// TIA Portal project "Parkplatz_1" (V20)

(* hardware
DEVICE "S7-1500/ET200MP-Station_1"  S7-1500 station
   slot 0: "Profilschiene_0"  Rack  6ES7 590-1***0-0AA0
   slot 1: "PLC_1"  CPU 1513-1 PN  6ES7 513-1AM03-0AB0  V4.0
      slot 3: "CPU-Display_1"  6ES7591-1AA00-0AA0
      slot 32768: "PROFINET-Schnittstelle_1"  X1
         slot 32769: "Port_1"  X1 P1
         slot 32770: "Port_2"  X1 P2
      slot 34817: "Virtual CP interface port_1"  Virtual CP interface port  Virtual CP interface port FW V4.0
   slot 2: "DI 16x24VDC BA_1"  DI 16x24VDC BA  6ES7 521-1BH10-0AA0  V1.1
   slot 3: "DQ 16x24VDC/0.5A ST_1"  DQ 16x24VDC/0.5A ST  6ES7 522-1BH00-0AB0  V2.0
   slot 4: "AI 8xU/I/R/RTD BA_1"  AI 8xU/I/R/RTD BA  6ES7 531-7QF00-0AB0  V1.0
   slot 5: "AQ 8xU/I HS_1"  AQ 8xU/I HS  6ES7 532-5HF00-0AB0  V2.2
   slot 6: "AQ 2xU/I ST_1"  AQ 2xU/I ST  6ES7 532-5NB00-0AB0  V1.0
*)

// ===== PLC "PLC_1"  CPU 1513-1 PN =====

VAR_GLOBAL   // PLC tag table "Standard-Variablentabelle"
   "PlcLabConnectIn01" AT %ID32760 : DWord;
   "PlcLabConnectIn02" AT %ID32764 : DWord;
   "PlcLabConnectOut01" AT %QD32760 : DWord;
   "PlcLabConnectOut02" AT %QD32764 : DWord;
   "Auto_rein_1" AT %M1.0 : Bool;
   "Auto_raus_1" AT %M1.1 : Bool;
   "Kein_Platz_frei" AT %M1.4 : Bool;
   "E1_Schranke_zu" AT %M2.0 : Bool;
   "A1_Schranke_zu" AT %M2.1 : Bool;
   "Plaetze_frei" AT %M1.5 : Bool;
   "Auto_raus_2" AT %M1.3 : Bool;
   "Auto_rein_2" AT %M1.2 : Bool;
   "E2_Schranke_zu" AT %M2.2 : Bool;
   "A2_Schranke_zu" AT %M2.3 : Bool;
END_VAR

VAR_GLOBAL   // PLC tag table "Eingänge"
   "B1" AT %E0.0 : Bool;   // Sensor 1 Einfahrt
   "B2" AT %E0.1 : Bool;   // Sensor 1 Ausfahrt
   "B3" AT %E0.2 : Bool;   // Sensor 2 Einfahrt
   "B4" AT %E0.3 : Bool;   // Sensor 2 Ausfahrt
   "S1" AT %E0.4 : Bool;   // Betriebsschalter
END_VAR

VAR_GLOBAL   // PLC tag table "Ausgänge"
   "P1" AT %A0.0 : Bool;   // Ampel 1 (rot)
   "P2" AT %A0.1 : Bool;   // Ampel 1 (grün)
   "P5" AT %AW32 : Int;   // Anzeige "Freie Parkplätze"
   "P6" AT %A0.4 : Bool;   // Schranke 1 Einfahrt
   "P7" AT %A0.5 : Bool;   // Schranke 1 Ausfahrt
   "P3" AT %A0.2 : Bool;   // Ampel 2 (rot)
   "P4" AT %A0.3 : Bool;   // Ampel 2 (grün)
   "P8" AT %A0.6 : Bool;   // Schranke 2 Einfahrt
   "P9" AT %A0.7 : Bool;   // Schranke 2 Ausfahrt
END_VAR

// folder: System blocks/Program resources

DATA_BLOCK "IEC_Counter_0_DB"   // DB1
{ S7_Optimized_Access := 'TRUE' }
AUTHOR : Simatic
FAMILY : IEC
NAME : CNTR
VERSION : 1.0
// stored: InstanceOfName IEC_COUNTER
"IEC_COUNTER"
BEGIN
   PV := 16;
END_DATA_BLOCK

DATA_BLOCK "IEC_Timer_0_DB"   // DB2
{ S7_Optimized_Access := 'TRUE' }
AUTHOR : Simatic
FAMILY : IEC
NAME : IEC_TMR
VERSION : 1.0
// stored: InstanceOfName IEC_TIMER
"IEC_TIMER"
BEGIN
END_DATA_BLOCK

DATA_BLOCK "IEC_Timer_0_DB_1"   // DB3
{ S7_Optimized_Access := 'TRUE' }
AUTHOR : Simatic
FAMILY : IEC
NAME : IEC_TMR
VERSION : 1.0
// stored: InstanceOfName IEC_TIMER
"IEC_TIMER"
BEGIN
END_DATA_BLOCK

DATA_BLOCK "IEC_Timer_0_DB_2"   // DB4
{ S7_Optimized_Access := 'TRUE' }
AUTHOR : Simatic
FAMILY : IEC
NAME : IEC_TMR
VERSION : 1.0
// stored: InstanceOfName IEC_TIMER
"IEC_TIMER"
BEGIN
END_DATA_BLOCK

DATA_BLOCK "IEC_Timer_0_DB_3"   // DB5
{ S7_Optimized_Access := 'TRUE' }
AUTHOR : Simatic
FAMILY : IEC
NAME : IEC_TMR
VERSION : 1.0
// stored: InstanceOfName IEC_TIMER
"IEC_TIMER"
BEGIN
END_DATA_BLOCK

// folder: (top level)

FUNCTION "Parkplatzsteuerung" : Void   // FC1, FBD
{ S7_Optimized_Access := 'TRUE' }
VERSION : 0.1
   VAR_TEMP   // added for the SCL form of the ladder/FBD networks
      _w1 : Bool;
      _w2 : Bool;
      _w3 : Bool;
      _w4 : Bool;
   END_VAR
BEGIN

REGION Network 1: Freie Plätze Zähler
   // Mithilfe des CTUD wird die Anzahl der freien Parkplätze gezählt. Über den Sensor B1 wird gezählt wenn ein Fahrzeug den Parkplatz betritt, dadurch gibt es einen freien Platz weniger. Über B2 wird gezählt wenn ein Fahrzeug den Parkplatz verlässt, dadurch gibt es einen freien Platz mehr. Die Grenze PV liegt auf 1, damit der Merker "Kein Platz frei" darunter auf FALSE geht. Bei 1 oder mehr gibt es freie Plätze, somit wird der Merker "Plätze frei" TRUE.
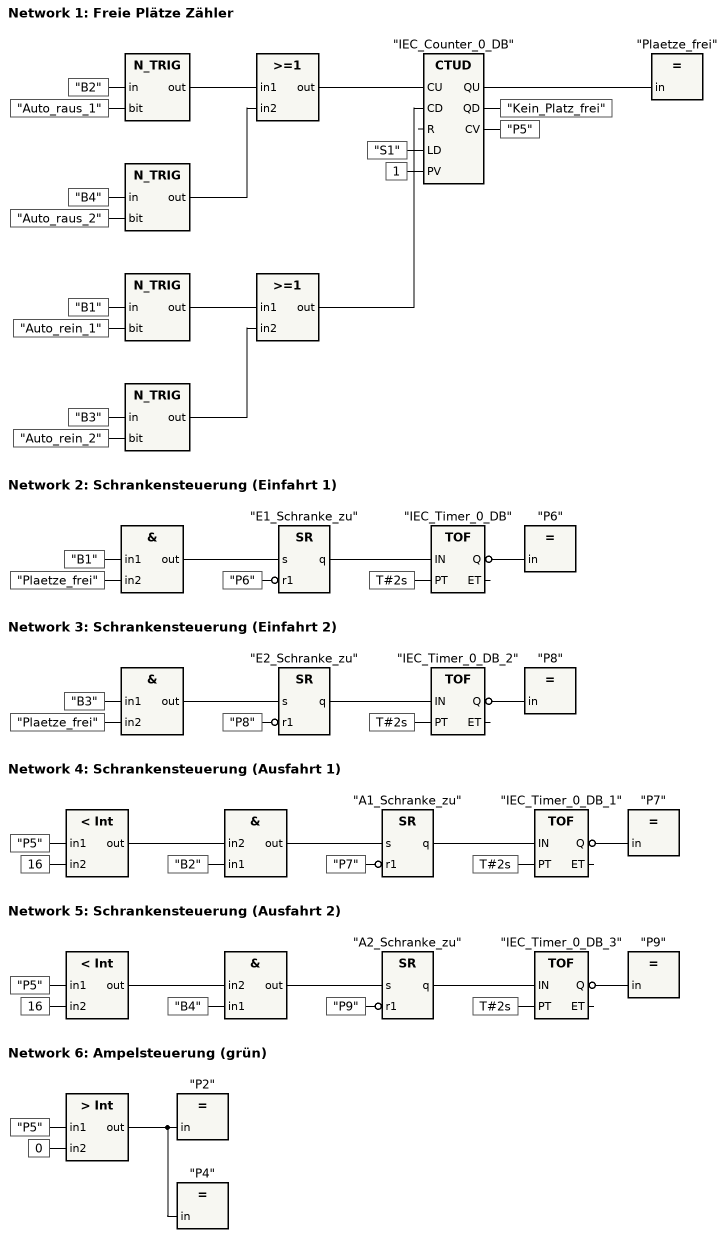
   #_w1 := NOT "B2" AND "Auto_raus_1";   // falling edge
   "Auto_raus_1" := "B2";
   #_w2 := NOT "B4" AND "Auto_raus_2";   // falling edge
   "Auto_raus_2" := "B4";
   #_w3 := NOT "B1" AND "Auto_rein_1";   // falling edge
   "Auto_rein_1" := "B1";
   #_w4 := NOT "B3" AND "Auto_rein_2";   // falling edge
   "Auto_rein_2" := "B3";
   "IEC_Counter_0_DB".CTUD(CU := #_w1 OR #_w2,
                           CD := #_w3 OR #_w4,
                           LD := "S1",
                           PV := 1,
                           QD => "Kein_Platz_frei",
                           CV => "P5");
   "Plaetze_frei" := "IEC_Counter_0_DB".QU;
END_REGION

REGION Network 2: Schrankensteuerung (Einfahrt 1)
   // Wenn ein Auto sich am Sensor befindet und noch Plätze frei sind, ermögliche die Einfahrt. Damit die Schranke dauerhaft geschlossen ist, wird der Ausgang der Ausschaltverzögerung dauerhaft negiert. Die Schranke öffnet also, wenn die Bedingung erfüllt ist und schließt dann nach 2s (nachdem das Auto eingefahren ist). Die Schranke setzt ihren Zustand selbst zurück.
   IF "B1" AND "Plaetze_frei" THEN
       "E1_Schranke_zu" := TRUE;   // SR flip-flop
   END_IF;
   IF NOT "P6" THEN "E1_Schranke_zu" := FALSE; END_IF;
   "IEC_Timer_0_DB".TOF(IN := "E1_Schranke_zu", PT := T#2s);
   "P6" := NOT "IEC_Timer_0_DB".Q;
END_REGION

REGION Network 3: Schrankensteuerung (Einfahrt 2)
   // Wenn ein Auto sich am Sensor befindet und noch Plätze frei sind, ermögliche die Einfahrt. Damit die Schranke dauerhaft geschlossen ist, wird der Ausgang der Ausschaltverzögerung dauerhaft negiert. Die Schranke öffnet also, wenn die Bedingung erfüllt ist und schließt dann nach 2s (nachdem das Auto eingefahren ist). Die Schranke setzt ihren Zustand selbst zurück.
   IF "B3" AND "Plaetze_frei" THEN
       "E2_Schranke_zu" := TRUE;   // SR flip-flop
   END_IF;
   IF NOT "P8" THEN "E2_Schranke_zu" := FALSE; END_IF;
   "IEC_Timer_0_DB_2".TOF(IN := "E2_Schranke_zu", PT := T#2s);
   "P8" := NOT "IEC_Timer_0_DB_2".Q;
END_REGION

REGION Network 4: Schrankensteuerung (Ausfahrt 1)
   // Wenn ein Auto sich am Sensor befindet und das Maximum an freien Plätze noch nicht erreicht ist, ermögliche die Ausfahrt. Damit die Schranke dauerhaft geschlossen ist, wird der Ausgang der Ausschaltverzögerung dauerhaft negiert. Die Schranke öffnet also, wenn die Bedingung erfüllt ist und schließt dann nach 2s (nachdem das Auto rausgefahren ist). Die Schranke setzt ihren Zustand selbst zurück.
   IF ("P5" < 16) AND "B2" THEN
       "A1_Schranke_zu" := TRUE;   // SR flip-flop
   END_IF;
   IF NOT "P7" THEN "A1_Schranke_zu" := FALSE; END_IF;
   "IEC_Timer_0_DB_1".TOF(IN := "A1_Schranke_zu", PT := T#2s);
   "P7" := NOT "IEC_Timer_0_DB_1".Q;
END_REGION

REGION Network 5: Schrankensteuerung (Ausfahrt 2)
   // Wenn ein Auto sich am Sensor befindet und das Maximum an freien Plätze noch nicht erreicht ist, ermögliche die Ausfahrt. Damit die Schranke dauerhaft geschlossen ist, wird der Ausgang der Ausschaltverzögerung dauerhaft negiert. Die Schranke öffnet also, wenn die Bedingung erfüllt ist und schließt dann nach 2s (nachdem das Auto rausgefahren ist). Die Schranke setzt ihren Zustand selbst zurück.
   IF ("P5" < 16) AND "B4" THEN
       "A2_Schranke_zu" := TRUE;   // SR flip-flop
   END_IF;
   IF NOT "P9" THEN "A2_Schranke_zu" := FALSE; END_IF;
   "IEC_Timer_0_DB_3".TOF(IN := "A2_Schranke_zu", PT := T#2s);
   "P9" := NOT "IEC_Timer_0_DB_3".Q;
END_REGION

REGION Network 6: Ampelsteuerung (grün)
   // Sobald Plätze frei sind (Zähler größer null), dann soll die Ampel grün leuchten.
   "P2" := "P5" > 0;
   "P4" := "P2";
END_REGION

REGION Network 7: Ampelsteuerung (rot)
   // Sobald keine Plätze mehr frei sind (Zähler kleiner eins), dann soll die Ampel rot leuchten.
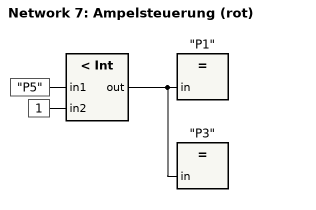
   "P1" := "P5" < 1;
   "P3" := "P1";
END_REGION
END_FUNCTION

ORGANIZATION_BLOCK "Main"   // OB1, FBD, ProgramCycle
TITLE = "Main Program Sweep (Cycle)"
{ S7_Optimized_Access := 'TRUE' }
VERSION : 0.1
   VAR_INPUT
      Initial_Call : Bool;   // Initial call of this OB
      Remanence : Bool;   // =True, if remanent data are available
   END_VAR
BEGIN

REGION Network 1
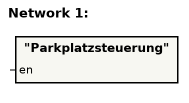
   "Parkplatzsteuerung"();
END_REGION
END_ORGANIZATION_BLOCK